FUNCTION_BLOCK DAC_RATE_LIMITER (* Basic FB with empty ECC *)
  (* Standard: 61499-2 *)
  (* Version 1.0, 2026-04-29, guilh *)
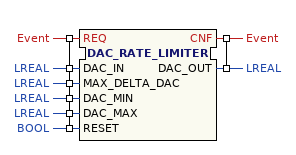
  EVENT_INPUT
    REQ WITH DAC_IN, MAX_DELTA_DAC, DAC_MIN, DAC_MAX, RESET;
  END_EVENT
  EVENT_OUTPUT
    CNF WITH DAC_OUT;
  END_EVENT
  VAR_INPUT
    DAC_IN : LREAL;
    MAX_DELTA_DAC : LREAL;
    DAC_MIN : LREAL;
    DAC_MAX : LREAL;
    RESET : BOOL;
  END_VAR
  VAR_OUTPUT
    DAC_OUT : LREAL;
  END_VAR
  VAR
    last_dac : LREAL;
    delta : LREAL;
    initialized : BOOL;
  END_VAR
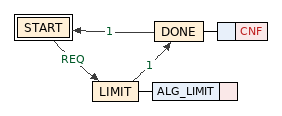
  EC_STATES
    START; (* Initial State *)
    LIMIT : ALG_LIMIT;
    DONE : -> CNF;
  END_STATES
  EC_TRANSITIONS
    START TO LIMIT := REQ;
    LIMIT TO DONE := 1;
    DONE TO START := 1;
  END_TRANSITIONS
  ALGORITHM ALG_LIMIT IN ST:
IF RESET THEN
    last_dac := DAC_IN;
    DAC_OUT := DAC_IN;
    initialized := TRUE;
ELSE
    IF NOT initialized THEN
        last_dac := DAC_IN;
        DAC_OUT := DAC_IN;
        initialized := TRUE;
    ELSE
        delta := DAC_IN - last_dac;

        IF delta > MAX_DELTA_DAC THEN
            DAC_OUT := last_dac + MAX_DELTA_DAC;
        ELSIF delta < -MAX_DELTA_DAC THEN
            DAC_OUT := last_dac - MAX_DELTA_DAC;
        ELSE
            DAC_OUT := DAC_IN;
        END_IF;

        IF DAC_OUT > DAC_MAX THEN
            DAC_OUT := DAC_MAX;
        ELSIF DAC_OUT < DAC_MIN THEN
            DAC_OUT := DAC_MIN;
        END_IF;

        last_dac := DAC_OUT;
    END_IF;
END_IF;
  END_ALGORITHM
END_FUNCTION_BLOCK
